Fanuc KAREL source: kx00019.KL

-- PROVISIONAL review KL for V940-1; original PC SHA256 32394212904f89b4d4a01299ed37a5a84e6630336aa053af573a8c1bfe5d9d7d
-- Incomplete behavior may be omitted. Consult companion uncertainty JSON. Do not deploy.
PROGRAM KX00019
%NOLOCKGROUP
VAR
  I : INTEGER
  J : INTEGER
  B : BOOLEAN
  F : FILE
  S : STRING[80]
-- UNRESOLVED_DECL P type=000102
-- UNRESOLVED_DECL SH type=002017
BEGIN
  -- V9_ZERO_TABLE_METADATA_HINT layout=0001; no indexed target words; source/name/runtime held
  -- UNRESOLVED_PC offsets 5-19; opcodes 2E,22,9D,33,B4
  -- UNRESOLVED_PC offsets 24-39; opcodes 22,9D,33,B3,23
  -- UNRESOLVED_PC offsets 44-48; opcodes 7F
END KX00019
